PROGRAM PRG_UnitTests
VAR
    fbWinchDemoTests : FB_WinchDemoTests;
END_VAR

fbWinchDemoTests();

END_PROGRAM

(* stored: Version 1.1.0.1
   POU PRG_UnitTests: Id {c5a7cd08-48ca-45cd-a7f2-11bb74cc6f7f}, SpecialFunc None *)
